INTERFACE ITF_SerialCommChannel

METHOD PUBLIC Send_String : Serial_FunctionResult
VAR_INPUT
	DATA	: STRING;	(*The string data to be sent to via the channel. Do not include the prefix/surfix.*)
END_VAR
END_METHOD

METHOD Fast_Task : Serial_FunctionResult
VAR_INPUT
END_VAR
END_METHOD

PROPERTY PREFIX : STRING
GET
END_GET
SET
END_SET
END_PROPERTY

PROPERTY SURFIX : STRING
SET
END_SET
GET
END_GET
END_PROPERTY

(*
	2015-06-04	:
		The method ReadString80(INT,STRING_PTR) should be used to read a string with a length of up to 80 characters long. 
*)
METHOD PUBLIC Read_String : Serial_FunctionResult
VAR_INPUT
	RECEIVED_DATA		: POINTER TO STRING;	(*The address of the variable to store the received string*)
END_VAR
END_METHOD

END_INTERFACE

(* stored: Version 1.1.0.1, ProductVersion 3.1.0.36
   Itf ITF_SerialCommChannel: Id {3d888eb0-87b4-4fa6-b61d-ac0bb3516463}
   Folder Properties: Id {5521f6d4-8bad-45a1-9562-319d3e2a4487}
   Folder Methods: Id {b582d091-adae-4ffd-bb10-3c067b46560b}
   Method Send_String: Id {0d4f238a-f17b-4743-af5a-72cb1e0ce69d}
   Method Fast_Task: Id {0e05445b-bbe6-452b-af95-a9eb0f551b35}
   Property PREFIX: Id {3b285f6a-a220-4e32-adeb-ae725137ed5b}
   Get Get: Id {4477abb0-1c66-44fd-8804-61ed8e286065}
   Set Set: Id {ce226e18-b994-4dfc-b636-e19d7f8569d7}
   Property SURFIX: Id {d47cad6f-e144-4db2-afa8-3c4b8fcbe262}
   Set Set: Id {2a37b684-2204-490e-9eef-ba81ade495e4}
   Get Get: Id {e38d0607-0a2b-4f90-99ce-db2524478468}
   Method Read_String: Id {f6935d50-15b2-4a13-b965-f6c201f0dc0f} *)
